Fanuc KAREL source: KA00172.KL

PROGRAM KA00172
%NOLOCKGROUP
VAR
  SRC: ARRAY[4] OF STRING[20]
  DST: ARRAY[4] OF INTEGER
BEGIN
  DST = SRC
END KA00172
